(* Logix 5000 project; controller Analog_Input Emulate 5570 rev 36.11; software revision 36.00 *)

TASK MainTask (continuous, watchdog 500 ms) : MainProgram, Emulation

MODULES
   Local : Emulate 5570 (ICP 2, rev 36.11)
       : 1756-IB16 (ICP 3, rev 3.1, Input RPI 20 ms)
       : vendor 1 type 7 code 16 (ICP 4, rev 3.1, Output RPI 20 ms)
       : 1756-IF8 (ICP 5, rev 1.1, Input RPI 100 ms)
END_MODULES

ADD_ON_INSTRUCTION Analog_In   (* revision 1.0 *)
VAR_INPUT
   Raw_Max : REAL; {required}   // Maximum Bit Balue
   Raw_Min : REAL; {required}
   EU_Max : REAL; {required}
   EU_Min : REAL; {required}
   Analog_Ch : REAL; {required}
END_VAR
VAR_OUTPUT
   EU_Value : REAL; {required}
END_VAR
VAR
   Analog : SCALE; {access None}   // Data Type for Add On Instruction
END_VAR

ROUTINE Logic   (* structured text *)
   Analog.In := Analog_Ch;
   Analog.InRawMax := Raw_Max;
   Analog.InRawMin := Raw_Min;
   Analog.InEUMax := EU_Max;
   Analog.InEUMin := EU_Min;
   SCL(Analog);
   EU_Value := Analog.Out;
END_ROUTINE
END_ADD_ON_INSTRUCTION

VAR_GLOBAL   (* controller tags *)
   CONVEYOR : ALIAS FOR Local:4:O.Data.0;   // Conveyor Motor
   ERROR : ALIAS FOR Local:4:O.Data.1;   // Part Feed Error Indicator
   HEIGHT : DINT;   // Scaled EU Value from Add On
   HEIGHT_SENSOR : ALIAS FOR Local:5:I.Ch0Data;   // Height Sensor for Add On
   PART_A : ALIAS FOR Local:3:I.Data.0;   // Part A N.O. Proximity Switch
   PART_A_ERROR : BOOL;   // Part A double part
   PART_A_UPPER : REAL;   // Part A Upper Limit
   PART_B : ALIAS FOR Local:3:I.Data.1;   // Part B N.O. Proximity Switch
   PART_B_ERROR : BOOL;   // Part B double part
   PART_B_UPPER : REAL;   // Part B Upper Limit
   RESET : ALIAS FOR Local:3:I.Data.2;   // RESET N.O. Pushbutton
   START : ALIAS FOR Local:3:I.Data.14;   // RESET N.O. Pushbutton
   STOP : ALIAS FOR Local:3:I.Data.15;   // STOP N.C. Pushbutton
END_VAR

PROGRAM Emulation   (* main routine Emulate *)
VAR
   emAIN_RESET : TIMER := (PRE := 3000);
   emCOUNT : COUNTER := (PRE := 6, ACC := 1);
   emCOUNT_PULSE : TIMER := (PRE := 6000, ACC := 96);
   emPART_A : BOOL;
   emPART_B : BOOL;
END_VAR

ROUTINE Emulate   (* ladder *)
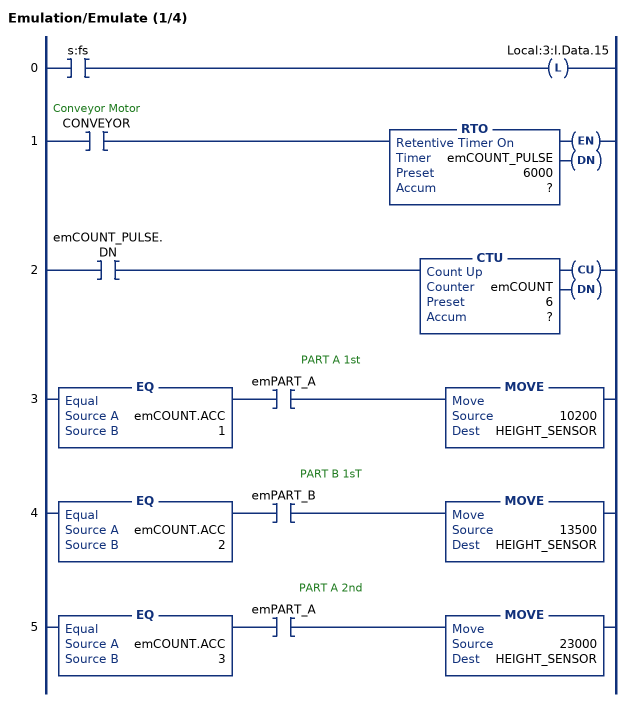
   0: XIC(s:fs)OTL(Local:3:I.Data.15);
   1: XIC(CONVEYOR)RTO(emCOUNT_PULSE,?,?);
   2: XIC(emCOUNT_PULSE.DN)CTU(emCOUNT,?,?);
   // PART A 1st
   3: EQ(emCOUNT.ACC,1)XIC(emPART_A)MOVE(10200,HEIGHT_SENSOR);
   // PART B 1sT
   4: EQ(emCOUNT.ACC,2)XIC(emPART_B)MOVE(13500,HEIGHT_SENSOR);
   // PART A 2nd
   5: EQ(emCOUNT.ACC,3)XIC(emPART_A)MOVE(23000,HEIGHT_SENSOR);
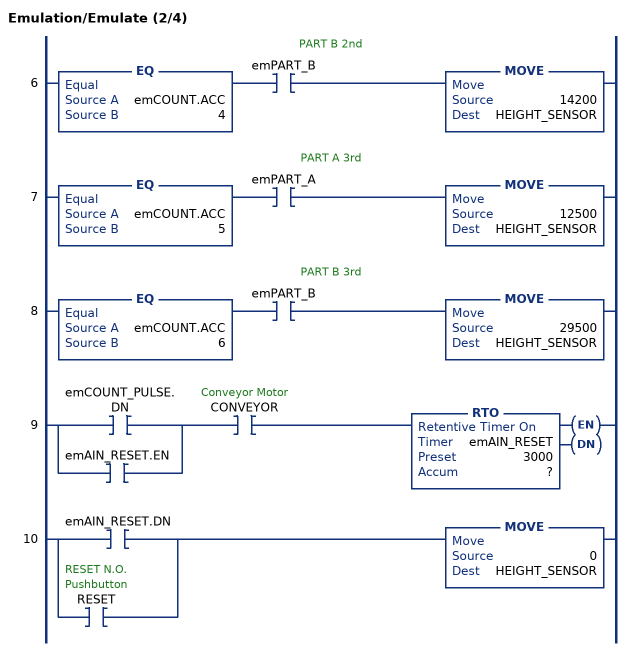
   // PART B 2nd
   6: EQ(emCOUNT.ACC,4)XIC(emPART_B)MOVE(14200,HEIGHT_SENSOR);
   // PART A 3rd
   7: EQ(emCOUNT.ACC,5)XIC(emPART_A)MOVE(12500,HEIGHT_SENSOR);
   // PART B 3rd
   8: EQ(emCOUNT.ACC,6)XIC(emPART_B)MOVE(29500,HEIGHT_SENSOR);
   9: [XIC(emCOUNT_PULSE.DN) ,XIC(emAIN_RESET.EN) ]XIC(CONVEYOR)RTO(emAIN_RESET,?,?);
   10: [XIC(emAIN_RESET.DN) ,XIC(RESET) ]MOVE(0,HEIGHT_SENSOR);
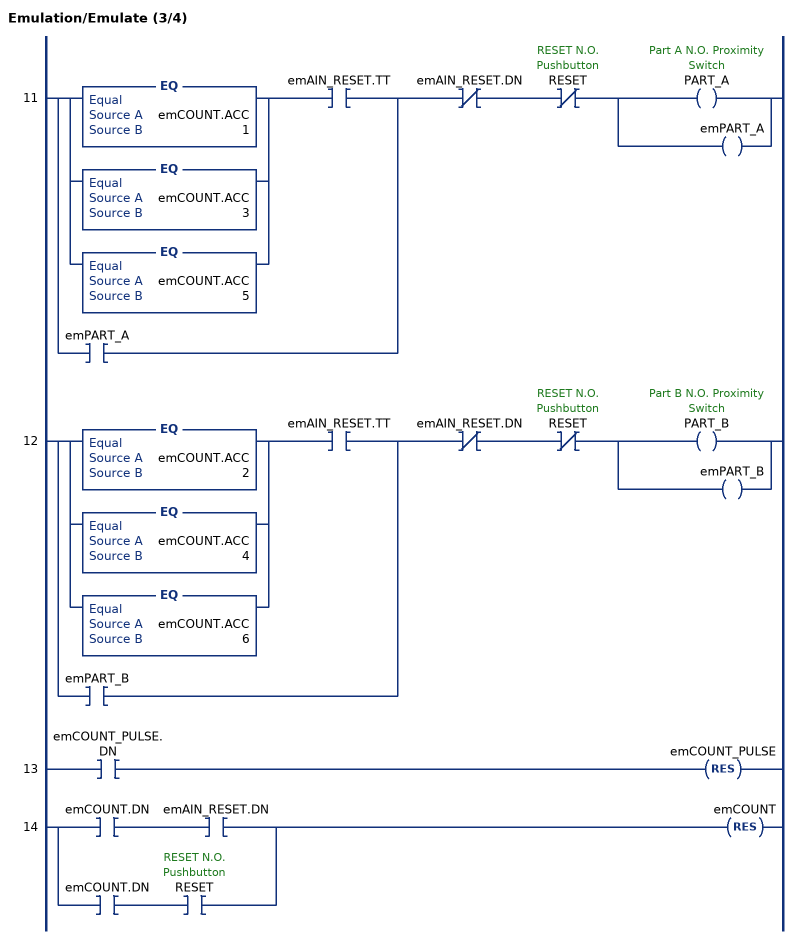
   11: [[EQ(emCOUNT.ACC,1) ,EQ(emCOUNT.ACC,3) ,EQ(emCOUNT.ACC,5) ] XIC(emAIN_RESET.TT) ,XIC(emPART_A) ]XIO(emAIN_RESET.DN)XIO(RESET)[OTE(PART_A) ,OTE(emPART_A) ];
   12: [[EQ(emCOUNT.ACC,2) ,EQ(emCOUNT.ACC,4) ,EQ(emCOUNT.ACC,6) ] XIC(emAIN_RESET.TT) ,XIC(emPART_B) ]XIO(emAIN_RESET.DN)XIO(RESET)[OTE(PART_B) ,OTE(emPART_B) ];
   13: XIC(emCOUNT_PULSE.DN)RES(emCOUNT_PULSE);
   14: [XIC(emCOUNT.DN) XIC(emAIN_RESET.DN) ,XIC(emCOUNT.DN) XIC(RESET) ]RES(emCOUNT);
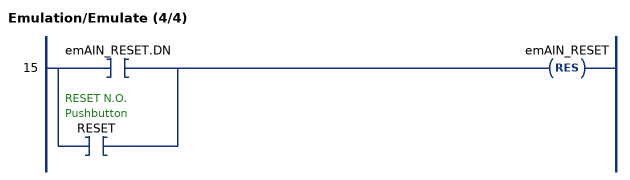
   15: [XIC(emAIN_RESET.DN) ,XIC(RESET) ]RES(emAIN_RESET);
END_ROUTINE
END_PROGRAM

PROGRAM MainProgram   (* main routine MainRoutine *)
VAR
   HEIGHT_SCALE : Analog_In := (Raw_Max := 32767.0, EU_Max := 100.0);   // Add On Instruction Tag for Analog Scalling
END_VAR

ROUTINE ConveyorControlRoutine   (* ladder *)
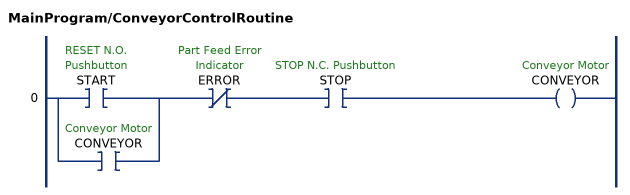
   0: [XIC(START) ,XIC(CONVEYOR) ]XIO(ERROR)XIC(STOP)OTE(CONVEYOR);
END_ROUTINE

ROUTINE MainRoutine   (* ladder *)
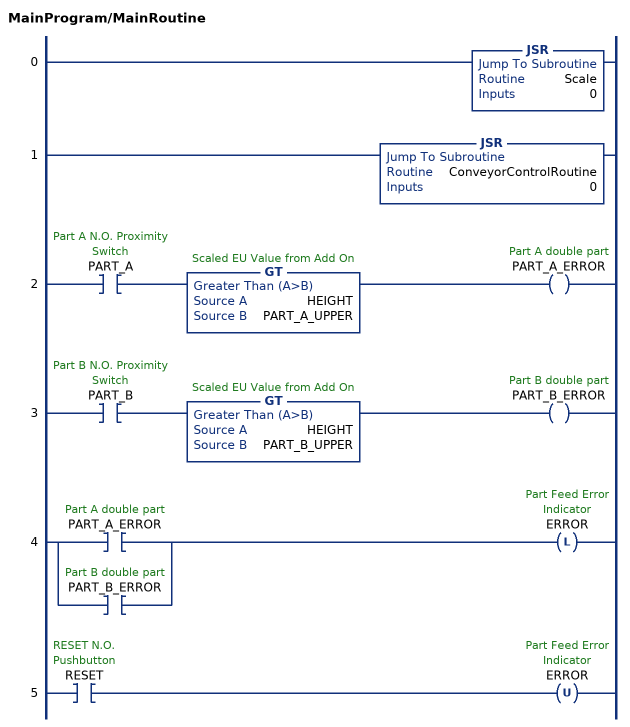
   0: JSR(Scale,0);
   1: JSR(ConveyorControlRoutine,0);
   2: XIC(PART_A)GT(HEIGHT,PART_A_UPPER)OTE(PART_A_ERROR);
   3: XIC(PART_B)GT(HEIGHT,PART_B_UPPER)OTE(PART_B_ERROR);
   4: [XIC(PART_A_ERROR) ,XIC(PART_B_ERROR) ]OTL(ERROR);
   5: XIC(RESET)OTU(ERROR);
END_ROUTINE

ROUTINE Scale   (* ladder *)
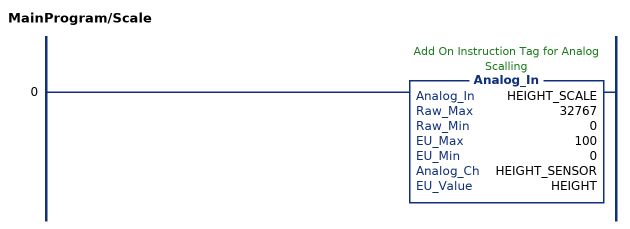
   0: Analog_In(HEIGHT_SCALE,32767,0,100,0,HEIGHT_SENSOR,HEIGHT);
END_ROUTINE
END_PROGRAM
